# EPICS SNL sequencer program: test/large_example.st
program example

%%#include <string.h>
%%#include <time.h>
%%#include <stdlib.h>
%%#include <stdio.h>

int myPv1;
assign myPv1 to "{PREFIX}:myPv1";
monitor myPv1;

int myPv2;
assign myPv2 to "{PREFIX}:myPv2";
monitor myPv2;

int myPv3;
assign myPv3 to "{PREFIX}:myPv3";
monitor myPv3;

int i=0;

ss state_set_1
{

    state state1

    {
		entry
		{
			myPv1=10;
			pvPut(myPv1);
		}

		when (myPv1==myPv2)
		{
			myPv1=0;
			myPv2=5;
		} state state2

		when (delay(4))
		{
			myPv1=5;
			if (myPv2==2) {
				myPv3+=3;
				myPv2=1;
			for (i=0; i<10; i++) {
				myPv1 += i;
				delay(5);
			}
			}
			else if (myPv2==3) {
				myPv3+=2;
			}
			else if (myPv2==3) {
				myPv3+=100;
			for (i=0; i<10; i++) {
				myPv1 += i;
				delay(5);
			}
			}
			else if (myPv2==3) {
				myPv3+=999;
			}
			myPv2 += 1;
		} state state3
	}

	state state2

	{
		when (    myPv2 < myPv3
			   && fabs( myPv2 - myPv1 ) > 5
			   || delay(1))
		{
			while (myPv2 < 10) {
				myPv2 += 1;
				delay(1);

			if (myPv1==5) {
				myPv1=4;
			}
			else if (myPv2==3) {
				myPv3+=333;
			}
			else {
				myPv1=3;
			}
			}
		} state state1

		when (delay(5) && (myPv2==5))
		{} state state3
	}

    state state3

    {
		when (myPv1>0)
		{} state state1

		when (myPv1==myPv2 || delay(3) && fabs( myPv3 - myPv1 ) < 3)
		{
			myPv1=0;
			for (i=0; i<10; i++) {
				myPv1 += i;
				delay(1);
			if (myPv1==5) {
				myPv1=4;
			while(myPv1<10){
				myPv2+=1;
			}
			}
			}

		} state state2
	}
}
